Universal Robots PolyScope program: Ruch3MS.urp

Program Ruch3MS (installation=default directory=/programs/usbdisk createdIn=3.15.8.106339 lastSavedIn=3.15.8.106339 robotSerialNumber=2020330428)
Calibrated DH parameters: a=[0.000029, -0.241913, -0.128453, -0.000049, -0.000012, 0]; d=[0.151842, -4.082088, 33.504745, -29.309875, 0.08529, 0.082285]; alpha=[1.571059, -0.006644, 0.005794, 1.571984, -1.571997, 0]; deltaTheta=[-0.000032, 0.111537, 0.813391, -0.924919, 0.000036, 0.000016]
Robot Program (runOnlyOnce=false)
  MoveJ speed 60 deg/s, acceleration 120 deg/s^2 (useActiveTCP=true)
    Waypoint Punkt_orienta_1: TCP in base x=-295.643 y=-272.772 z=394.537 mm, rx=1.2032 ry=1.2167 rz=-1.1995 rad; joints [0, -90, 90, -90, -0.003, 0] deg; flange x=-296.484 y=-197.777 z=394.765 mm, rx=1.2032 ry=1.2167 rz=-1.1995 rad
    Waypoint Punkt_orienta_2: TCP in base x=299.32 y=-268.848 z=396.261 mm, rx=1.2077 ry=-1.2055 rz=1.2126 rad; joints [0.003, -89.999, -90, -89.997, 0, 0.004] deg; flange x=299.171 y=-193.848 z=395.967 mm, rx=1.2077 ry=-1.2055 rz=1.2126 rad
